*)
(* EXIT the routine IF it was executed the 10 seconds which is equal to 0.04 degrees accuracy *)
IF T_PLC_MS() - last < 10000 THEN RETURN; END_IF;
last := T_PLC_MS();

(* calculate the angles *)
N := DWORD_TO_REAL(DT_TO_DWORD(utc) - 946728000)/86400;
LA := RAD(latitude);
SLA := SIN(LA);
CLA := COS(LA);
LO := Rad(longitude);
L := modR(280.460 + 0.9856474 * N,360);
G := Rad(modR(357.528 + 0.9856003 * N,360));
K := Rad(L + 1.915 * SIN(G) + 0.02 * SIN(2*G));
X := Rad(23.439 - 0.0000004 * N);
A := ATAN(COS(X)*TAN(K));
IF COS(K) < 0 THEN A := A + PI1; END_IF;
D := ASIN(SIN(X) * SIN(K));
TA := RAD(MODR(6.697376 + 0.065709825 * DINT_TO_REAL(TRUNC(N - 0.5)) + 0.5 + TOD_TO_REAL(DT_TO_TOD(utc)) * 2.78538333E-7, 24) * 15 + longitude - DEG(A));
CTA := COS(TA);
T1 := CTA*SLA - TAN(D)*CLA;
B := deg(ATAN(SIN(TA)/T1));
IF T1 < 0 THEN B := B + 180; END_IF;
IF B > 180 THEN
	B := B - 180;
ELSIF B < 180 THEN
	B := B + 180;
END_IF;
H := deg(ASIN(COS(D)*CTA*CLA+SIN(D)*SLA));
HR := H + 0.017 / TAN(Rad(H+10.3/(H+5.11)));


(* revision history
hm	1. feb 2007	rev 1.0
	original version

hm	6. jan 2008	rev 1.1
	performance improvements

hm	18. jan 2008	rev 1.2
	further performance improvements
	only calculate once every 10 seconds

hm	16. mar. 2008	rev 1.3
	added type conversion to avoid warnings under codesys 3.0

hm	30. jun. 2008	rev 1.4
	added type conversions to avoid warnings under codesys 3.0

*)
END_FUNCTION_BLOCK

(* POU SUN_TIME, ST *)
FUNCTION_BLOCK SUN_TIME
VAR_INPUT
	latitude : REAL;				(* latitude of geographical position  *)
	longitude : REAL;				(* longitude of geographical position  *)
	utc : DT;						(*	world time				*)
END_VAR
VAR_OUTPUT
	sun_midday : TOD;			(*	astrological midday in hours when sun stand at south direction	*)
	sun_rise : TOD;				(*	sun rise for current day in local time *)
	sun_set : TOD;				(*	sun set for current day in local time *)
	sun_declination : REAL;		(*	sun declination at midday in degrees	*)
END_VAR
VAR
	T: INT;							(* day in the year   *)
	DK: REAL;						(* sun declination at midday *)
	delta: REAL;					(* delta from midday for sunrise and sunset  *)
	h: REAL;
	B: REAL;
	offset : REAL;
	l15: REAL;
	dat: DATE;
	last_dat: DATE;
END_VAR

(*
version 1.4	17. jan 2008
programmer 	hugo
tested by	tobias

this FUNCTION block calculates the sun rise, sun set, sun offset at midday sun declination for a given date 
for performance reasons the algorithm has been simplified and is accurate within a few minutes only 
the times are calculated in utc and have to be corrected for the given time zone
this correction is not done within sun_time because it would be a problem on days where dst is enabled or disabled


*)
dat := DT_TO_DATE(utc);
IF dat = last_dat THEN RETURN; END_IF;
last_dat := dat;
l15 := longitude * 0.0666666666666;
B := latitude * 0.0174532925199433;
h := -0.0145;
T := day_of_year(dat);
offset := -0.1752 * SIN(0.033430*T + 0.5474) - 0.1340*SIN(0.018234*T - 0.1939);
sun_midday := hour_to_tod(12 + Offset - l15);
DK := 0.40954 * SIN(0.0172 * (T-79.35));
sun_declination := deg(DK);
delta := 12*ACOS((SIN(h) - SIN(B) * SIN(DK)) / (COS(B) * COS(DK))) * 0.318309886;
sun_rise := hour_to_tod(12 - delta - Offset - l15);
sun_set := hour_to_tod(12 + delta - Offset - l15);

(* revision history

rev 1.1	hm	20.1.2007
	deleted unused variables sun_riseR and sun_setR

rev 1.2 hm 17.4.2007
	corrected error while sun:midday would not be corrected for longitude.

rev 1.3	hm	6. jan 2008
	performance improvements

rev	1.4 hm	17. jan 2008
	calculation is now only performed once a day
*)
END_FUNCTION_BLOCK

(* POU SWAP_BYTE, ST *)
FUNCTION SWAP_BYTE : WORD
VAR_INPUT
	IN : WORD;
END_VAR
VAR
END_VAR

(*
version 1.0	4 feb 2008
programmer 	hugo
tested by		tobias

This function swaps the high and low byte of the word in.

*)
Swap_Byte := ROL(in,8);


(* revision history
hm		4. feb 2008	rev 1.0
	original version

*)
END_FUNCTION

(* POU SWAP_BYTE2, ST *)
FUNCTION SWAP_BYTE2 : DWORD
VAR_INPUT
	IN : DWORD;
END_VAR
VAR
END_VAR

(*
version 1.0	4 feb 2008
programmer 	hugo
tested by		tobias

This function reverses the byte order in the dword.

*)
Swap_Byte2 := (ROR(in,8) AND 16#FF00FF00) OR (ROL(in,8) AND 16#00FF00FF);

(* revision history
hm		4. feb 2008	rev 1.0
	original version

*)
END_FUNCTION

(* POU SWITCH_I, ST *)
FUNCTION_BLOCK SWITCH_I
VAR_INPUT
	set : BOOL;
	in : BOOL;
	rst : BOOL;
END_VAR
VAR_INPUT CONSTANT
	T_debounce : TIME := T#10ms;
	T_reconfig : TIME := T#1s;
	T_on_max : TIME := T#0h;
END_VAR
VAR_OUTPUT
	Q : BOOL := 0;
END_VAR
VAR
	state : BYTE := 0;
	edge : BOOL := 0;
	r_edge : BOOL := 0;
	T_on : TIME;
	tx: TIME;
END_VAR

(*
version 1.1	15 sep 2007
programmer 	oscat
tested by		tobias

this is an intelligent switch interface which has an autodetect feature for in and it will detect the type of switch connected automatically
the input can be connected to low active pulses, high active pulses and on/off switch.
it will automatically adjust to the correct type without manual adjustment
a configurable debounce timer will debounce input signals
if t_on_max is set to anything other then 0 the output will be turned off after the max on time is reached.

*)
(* read system time *)
tx := DWORD_TO_TIME(T_PLC_MS());

(* asynchronous set and reset first *)
IF set AND NOT rst THEN
	Q := 1;
	T_on := tx;
ELSIF rst THEN
	Q := 0;
(* check FOR input edge AND start debounce timer *)
ELSIF (in XOR edge) AND NOT (state = 1) THEN
	state := 1;
	T_on := Tx;
(* edge was detected and debounce time elapsed *)
ELSIF (state = 1) AND (Tx - t_debounce >= T_on) THEN
	state := 2;
	(* react on rising or falling edge depending on r_edge *)
	IF r_edge XOR in THEN Q := NOT Q; END_IF;
(* wait for T_reconfig and adjust r_edge *)
ELSIF state = 2 AND Tx - t_reconfig >= T_on THEN
	r_edge := in;
END_IF;
IF Q AND T_on_max > t#0ms AND Tx >= T_on + T_on_max THEN
	Q := FALSE;
END_IF;
edge := in;

(* revision history

hm	4 aug 2006	rev 1.0
	original version

hm	15.9.2007	rev 1.1
	replaced Time() with T_PLC_MS for compatibility and performance reasons

*)
END_FUNCTION_BLOCK

(* POU SWITCH_X, ST *)
FUNCTION_BLOCK SWITCH_X
VAR_INPUT
	IN1 : BOOL;
	IN2 : BOOL;
	IN3 : BOOL;
	IN4 : BOOL;
	IN5 : BOOL;
	IN6 : BOOL;
END_VAR
VAR_OUTPUT
	Q1 : BOOL;
	Q2 : BOOL;
	Q3 : BOOL;
	Q4 : BOOL;
	Q5 : BOOL;
	Q6 : BOOL;
	Q31 : BOOL;
	Q41 : BOOL;
	Q51 : BOOL;
	Q61 : BOOL;
	Q32 : BOOL;
	Q42 : BOOL;
	Q52 : BOOL;
	Q62 : BOOL;
END_VAR
VAR_INPUT CONSTANT
	t_debounce : TIME := t#50ms;
END_VAR
VAR
	init : BOOL;
	T1, T2, T3, T4, T5, T6 : TOF;
	tx: TIME;
	x1: BOOL;
	x2: BOOL;
	E1, E2 : BOOL;
END_VAR

(*
version 1.0	15 Feb 2007
programmer 	oscat
tested by		tobias

*)
(* initialize on startup *)
IF NOT init THEN
	init := TRUE;
	IF t_debounce < t#50ms THEN tx := t#50ms; ELSE tx := t_debounce; END_IF;
	T1(PT := Tx);
	T2(PT := Tx);
	T3(PT := Tx);
	T4(PT := Tx);
	T5(PT := Tx);
	T6(PT := Tx);
ELSE
	Q1 := FALSE;
	Q2 := FALSE;
	Q3 := FALSE;
	Q4 := FALSE;
	Q5 := FALSE;
	Q6 := FALSE;
	Q31 := FALSE;
	Q41 := FALSE;
	Q51 := FALSE;
	Q61 := FALSE;
	Q32 := FALSE;
	Q42 := FALSE;
	Q52 := FALSE;
	Q62 := FALSE;
END_IF;

(* read inputs and debounce *)
	T1(IN := IN1);
	T2(IN := IN2);
	T3(IN := IN3);
	T4(IN := IN4);
	T5(IN := IN5);
	T6(IN := IN6);

(* detect edge of IN1 and IN2 *)
IF t1.Q AND NOT E1 THEN X1 := TRUE; END_IF;
IF t2.Q AND NOT E2 THEN X2 := TRUE; END_IF;

IF t1.Q THEN
	IF t3.q THEN
		q31 := TRUE;
		X1 := FALSE;
	ELSIF t4.q THEN
		q41 := TRUE;
		X1 := FALSE;
	ELSIF t5.q THEN
		q51 := TRUE;
		X1 := FALSE;
	ELSIF t6.q THEN
		q61 := TRUE;
		X1 := FALSE;
	END_IF;
ELSIF t2.Q THEN
	IF t3.q THEN
		q32 := TRUE;
		X2 := FALSE;
	ELSIF t4.q THEN
		q42 := TRUE;
		X2 := FALSE;
	ELSIF t5.q THEN
		q52 := TRUE;
		X2 := FALSE;
	ELSIF t6.q THEN
		q62 := TRUE;
		X2 := FALSE;
	END_IF;
(* in1 was active alone *)
ELSIF NOT T1.Q AND E1 AND X1 THEN
	Q1 := TRUE;
	X1 := FALSE;
ELSIF NOT T2.Q AND E2 AND X2 THEN
	Q2 := TRUE;
	X2 := FALSE;
ELSIF T3.Q THEN
	Q3 := TRUE;
ELSIF T4.Q THEN
	Q4 := TRUE;
ELSIF T5.Q THEN
	Q5 := TRUE;
ELSIF T6.Q THEN
	Q6 := TRUE;
END_IF;

(* save state of in1 and in2 *)
E1 := T1.Q;
E2 := T2.Q;
END_FUNCTION_BLOCK

(* POU TANH, ST *)
FUNCTION TANH : REAL
VAR_INPUT
	X : REAL;
END_VAR
VAR
END_VAR


(*
version 1.2	10. mar 2008
programmer 	hugo
tested by	tobias

this function calculates the tangens hyperbolicus

*)
IF X > 20 THEN
	tanH := 1;
ELSIF X < -20 THEN
	tanH := -1;
ELSE
	tanH := 1 - 2 / (EXP(2 * x) + 1);
END_IF;

(* revision hisdtory
hm		12.1.2007		rev 1.0
	original version

hm		1.12.2007		rev 1.1
	changed code to improve performance

hm		10. mar 2008	rev 1.2
	corrected an error in formula
	extended range of valid inputs to +/- INV
*)
END_FUNCTION

(* POU TANK_LEVEL, ST *)
FUNCTION_BLOCK TANK_LEVEL
VAR_INPUT
	LEVEL : BOOL;
	LEAK : BOOL;
	ACLR : BOOL;
END_VAR
VAR_INPUT CONSTANT
	MAX_VALVE_TIME : TIME := T#0s;
	LEVEL_DELAY_TIME : TIME := T#0s;
END_VAR
VAR_OUTPUT
	VALVE : BOOL;
	ALARM : BOOL;
	STATUS : BYTE;
END_VAR
VAR
	cx : ACTUATOR_COIL;
	tn : TON;
	tl : TONOF;
	open: BOOL;
END_VAR


(*
version 1.0	27 feb 2007
programmer 	hugo
tested by		tobias

*)
(* preprocess the level information *)
tl(in := level, T1 := level_delay_time, T2 := level_delay_time);
open := tl.Q;

(* start logic *)
IF ALARM THEN
	(* check for ACLR if ALARM is present *)
	IF ACLR THEN
		ALARM := FALSE;
		STATUS := 101; (* aclr pressed *)
		cx(in := FALSE);
	END_IF;
	RETURN;
ELSIF LEAK THEN
	(* leakeage detected *)
	cx(in := FALSE);
	ALARM := TRUE;
	STATUS := 1;	(* leakeage error *)
ELSIF open THEN
	(* valve needs to be opened because level is too low *)
	cx(in := TRUE);
	STATUS := 102; (* valve open by low level *)
ELSE
	(* valve needs to be closed *)
	cx(in := FALSE);
	STATUS := 100; (* valve idle *)
END_IF;

(* check if valve is open too long and generate alarm if necessary *)
tn(in := cx.out AND (MAX_VALVE_TIME > T#0s), PT := MAX_VALVE_TIME);
IF tn.Q THEN
	ALARM := TRUE;
	STATUS := 2; (* overtime error *)
	cx(in := FALSE);
END_IF;

(* set output signal *)
VALVE := cx.out;
END_FUNCTION_BLOCK

(* POU TONOF, ST *)
FUNCTION_BLOCK TONOF
VAR_INPUT
	IN : BOOL;
	T1, T2 : TIME;
END_VAR
VAR_OUTPUT
	Q : BOOL;
END_VAR
VAR
	X : TON;
	Y : TOF;
END_VAR

(*
version 1.1	17 sep 2007
programmer 	hugo
tested by		tobias

TONOF generated a TON and TOF Delay for the Input N TON (T1) and TOF (T2) can be configured separately
*)
X(IN := IN, PT := T1);
Y(in := X.Q, PT := T2);
Q := Y.Q;

(* revision history
hm	10. dec 2007	rev 1.0
	original version

*)
	
END_FUNCTION_BLOCK

(* POU TC_MS, ST *)
FUNCTION_BLOCK TC_MS
VAR_INPUT
END_VAR
VAR_OUTPUT
	TC : DWORD;
END_VAR
VAR
	init: BOOL;
	tx: DWORD;
	last: DWORD;
END_VAR

(*
	version 1.0	13 mar 2008
	programmer 	hugo
	tested by		tobias

TC_MS delivers the time it was last called on the output TC in Milliseconds.

*)
(* read system timer *)
tx := T_PLC_MS();

IF NOT init THEN
	init := TRUE;
	TC := 0;
ELSE
	tc := tx - last;
END_IF;
last := tx;

(* revision history
hm		13. mar. 2008	rev 1.0
	original version

*)
END_FUNCTION_BLOCK

(* POU TC_US, ST *)
FUNCTION_BLOCK TC_US
VAR_INPUT
END_VAR
VAR_OUTPUT
	TC : DWORD;
END_VAR
VAR
	init: BOOL;
	tx: DWORD;
	last: DWORD;
END_VAR

(*
	version 1.0	13 mar 2008
	programmer 	hugo
	tested by		tobias

TC_US delivers the time it was last called on the output TC in Microseconds.

*)
(* read system timer *)
tx := T_PLC_US();

IF NOT init THEN
	init := TRUE;
	TC := 0;
ELSE
	tc := tx - last;
END_IF;
last := tx;

(* revision history
hm		13. mar. 2008	rev 1.0
	original version

*)
END_FUNCTION_BLOCK

(* POU TEMP_EXT, ST *)
FUNCTION_BLOCK TEMP_EXT
VAR_INPUT
	t_ext1 : REAL;
	t_ext2 : REAL;
	t_ext3 : REAL;
	t_ext_config : BYTE := 0;
	dt_in : DT;
END_VAR
VAR_INPUT CONSTANT
	t_ext_min : REAL := -40;
	t_ext_max : REAL := 60;
	t_ext_default : REAL := -10;
	heat_period_start : DATE := D#1970-9-1;
	heat_period_stop : DATE := D#1970-4-30;
	cool_period_start : DATE := D#1970-4-1;
	cool_period_stop : DATE := D#1970-9-30;
	heat_start_temp_day : REAL := 15;
	heat_start_temp_night : REAL := 10;
	heat_stop_temp : REAL := 18;
	cool_start_temp_day : REAL := 26;
	cool_start_temp_night : REAL := 26;
	cool_stop_temp : REAL := 24;
	start_day : TOD := tod#09:00;
	start_night : TOD := tod#21:00;
	cycle_time : TIME := t#10m;
END_VAR
VAR_OUTPUT
	t_ext : REAL;
	heat : BOOL;
	cool : BOOL;
END_VAR
VAR
	tx: TIME;
	last_run: TIME;
	init: BOOL;
	cool_start: DATE;
	cool_stop: DATE;
	heat_start: DATE;
	heat_stop: DATE;
	xdate: DATE;
	day: BOOL;
END_VAR


(*
version 1.1	15 sep 2007
programmer 	hugo
tested by		tobias

temp_ext measures and processes ext temperature and decides if heating or cooling is needed.

 the measurement of t_ext has 3 inputs which can be configured in different ways:
	t_ext_config = 0 means the ext temp is the avg of the 3 external temperatures, this mode is the default mode.
	t_ext_config = 1 means t_ext1 is used.
	t_ext_config = 2 means t_ext1 is used.
	t_ext_config = 3 means t_ext1 is used.
	t_ext_config = 4 means t_ext_default is used.
	t_ext_config = 5 means the lowest of the 3 external temperatures is used.
	t_ext_config = 6 means the higest externnal temperature is used.
	t_ext_config = 7 means the midlle external temperature is used, if there are only two working, the lowest is used.
	in any config mode, an external temperature higher then t_ext_max or lower then t_ext_min is ignored to prevent from temperatures caused by broken sensors or wires.
	if no external temperature is available, a default value (t_ext_default) is used.
	if you have only one external sensor, connect the 3 inputs to the same sensor, or select the right input with t_ext_config.

heating or cooling is enabled during heating / cooling period when the day or night start temperature is reached for at least the specified delay time and will be disabled after the stop temperature is reached. 
t_ext output can be used by other modules to determine the correct system temperature for heating or cooling.

*)
IF NOT init THEN
	init := TRUE;
	heat_start := set_Date(1972,month(heat_period_start),day_of_month(heat_period_start));
	heat_stop := set_Date(1972,month(heat_period_stop),day_of_month(heat_period_stop));
	cool_start := set_Date(1972,month(cool_period_start),day_of_month(cool_period_start));
	cool_stop := set_Date(1972,month(cool_period_stop),day_of_month(cool_period_stop));
END_IF;

(* read system time *)
tx := DWORD_TO_TIME(T_PLC_MS());

(* for efficiency exit isf this program has been executed less then 1min ago *)
IF tx - last_run < cycle_time THEN RETURN; END_IF;

(* calculate frequently used variables *)
xdate := set_Date(1972,month(DT_TO_DATE(dt_in)),day_of_month(DT_TO_DATE(dt_in)));
day := DT_TO_TOD(dt_in) >= start_day AND  DT_TO_TOD(dt_in) < start_night;

(* read the correct external temperature depending on the t_ext_config setting *)
t_ext := multi_in(t_ext1, t_ext2, t_ext3, t_ext_default, t_ext_min, t_ext_max, t_ext_config);

(* dtermine heating *)
IF (heat_start <= heat_stop AND xdate >= heat_start AND xdate <= heat_stop) OR (heat_start > heat_stop AND (xdate >= heat_start OR xdate <= heat_stop)) THEN
	(* heating period id true check for temperature *)
	IF day AND t_ext <= heat_start_temp_day THEN
		heat := TRUE;
	ELSIF NOT day AND t_ext <= heat_start_temp_night THEN
		heat := TRUE;
	ELSIF t_ext >= heat_stop_temp THEN
		heat := FALSE;
	END_IF;
ELSE
	heat := FALSE;
END_IF;

(* dtermine cooling *)
IF (cool_start <= cool_stop AND xdate >= cool_start AND xdate <= cool_stop) OR (cool_start > cool_stop AND (xdate >= cool_start OR xdate <= cool_stop)) THEN
	(* cooling period is true check for temperature *)
	IF day AND t_ext >= cool_start_temp_day THEN
		cool := TRUE;
	ELSIF NOT day AND t_ext >= cool_start_temp_night THEN
		cool := TRUE;
	ELSIF t_ext <= cool_stop_temp THEN
		cool := FALSE;
	END_IF;
ELSE
	cool := FALSE;
END_IF;

last_run := tx;

(* revision history
hm	6 dec 2006		rev 1.0
	original version

hm	15.9.2007		rev 1.1
	replaced Time() with T_PLC_MS for compatibility and performance reasons

*)
END_FUNCTION_BLOCK

(* POU TEMP_NI, ST *)
FUNCTION TEMP_NI : REAL
VAR_INPUT
	Res : REAL;
	R0 : REAL;
END_VAR
VAR
END_VAR

(*
version 1.4	6. Jan 2008
programmer 	hugo
tested by		tobias

this function returns the temperature for a nickel sensor in a range from -60..+180 °C *)
Temp_NI := (SQRT(0.30085225 - 2.66E-3 * (R0 - Res)) - 0.5485) * 751.8796992;

(*Temp_NI := 60;
WHILE step > accuracy DO
	IF Res_NI(Temp_NI,R0) < res THEN Temp_NI := Temp_NI + step; ELSE Temp_NI := Temp_NI - step; END_IF;
	step := step / 2;
END_WHILE;
*)
(* code before rev 1.3
Temp_NI := -60.0;
WHILE step > accuracy DO
	(* test if result greater or less *)
	IF Res_NI(Temp_NI + step,R0) < res THEN Temp_NI := Temp_NI + step; END_IF;
	step := step / 2;
END_WHILE;
*)

(* revision history

rev 1.1 	hm 24.1.2007	
	deleted unused variable A, B, C

rev 1.2		hm 10.9.2007
	changed accuracy to 0.02 degrees to improove performace

hm 17. 12 2007		rev 1.3
	improovements for better performance and higher accuracy

hm	6. jan 2008		rev 1.4
	further performance improvement
*)
END_FUNCTION

(* POU TEMP_PT, ST *)
FUNCTION TEMP_PT : REAL
VAR_INPUT
	Res : REAL;
	R0 : REAL;
END_VAR
VAR CONSTANT
	A : REAL := 3.9083E-3 ;
	B : REAL := -5.775E-7;
	accuracy : REAL := 0.02;
END_VAR
VAR
	step: REAL := 50.0;
	X: REAL;
	Y: REAL;
	t1: REAL;
END_VAR

(*
version 1.5	5. jan 2008
programmer 	hugo
tested by		tobias

this function returs the temperature for a platinum sensor for a range from -200..+850 °C *)
X := A * R0;
Y := B * R0;
IF Res >= R0 THEN
	t1 := X*X-4*Y*(R0-Res);
	IF t1 < 0 THEN
		Temp_PT := 10000;
	ELSE
		Temp_PT := (-X + SQRT(t1)) / (2 * Y);
	END_IF;
ELSE
	(* since the formula cannot be solved this is a successive approximation *)
	Temp_PT := -100.0;
	WHILE step > accuracy DO
		(* test if result greater or less *)
		IF Res_PT(Temp_PT,R0) < res THEN Temp_PT := Temp_PT + step; ELSE Temp_PT := Temp_PT - step; END_IF;
		step := step * 0.5;
	END_WHILE;
END_IF;

(* revision history

rev 1.1 hm 24.1.2007	
	deleted unused variable C

rev 1.2 hm 10.9.2007
	reduced accuracy to 0.02 to shorten execution time

rev 1.3	hm	2. dec 2007
	changed code for better performance

rev	1.4	hm	23. dec 2007
	avoid a negative square root if input values are wrong

rev 1.5 hm	5. jan 2008
	replaced / 2 with * 0.5 for better performance
*)
END_FUNCTION

(* POU TEMP_SI, ST *)
FUNCTION TEMP_SI : REAL
VAR_INPUT
	Res : REAL;
	RS : REAL;
	TS : REAL;
END_VAR
VAR CONSTANT
END_VAR
VAR
END_VAR

(*
version 1.4	6. jan 2008
programmer 	hugo
tested by		tobias

this function returs the temperature for a silicon sensor for a range from -60..+180 °C
for example KTY10 RS at TS normally 25 °C
*)
Temp_SI := (-7.64E-3 + SQRT(Res/RS* 6.64E-5 - 0.803E-5)) * 30120.48193 + TS;

(* code before rev 1.3
Temp_SI := -60;
WHILE step > accuracy DO
	(* test if result greater or less *)
	IF Res_SI(Temp_SI + step,RS,TS) < Res THEN Temp_SI := Temp_SI + step; END_IF;
	step := step / 2;
END_WHILE;
*)

(* revision history

hm 24.1.2007		rev 1.1
	the function would only work for TS = 25, now it works for other values of ts.

hm 10.9.2007		rev 1.2
	changed the function to use successive approcimation to avoid an error generated by a sqrt from a negative result.
	changed accuracy to 0.02 degrees to shorten execution time

hm 17. 12 2007		rev 1.3
	improovements for better performance

hm	6. jan 2008		rev 1.4
	further performance improvement
*)
END_FUNCTION

(* POU TEMPERATURE, ST *)
FUNCTION_BLOCK TEMPERATURE
VAR_INPUT
	K : REAL;
	C : REAL := -273.15;
	F : REAL := -459.67;
	Re : REAL := -218.52;
	Ra : REAL := 0;
END_VAR
VAR_OUTPUT
	YK : REAL;
	YC : REAL;
	YF : REAL;
	YRe : REAL;
	YRa : REAL;
END_VAR
VAR
END_VAR

(*
version 1.0	21 feb 2008
programmer 	hugo
tested by	oscat

this function converts different temperature units
any unused input can simply be left open.
different inputs connected at the same time will be added up.

*)
YK := K + (C + 273.15) + (F + 459.67) * 0.555555555555 + (Re * 1.25 + 273.15) + (Ra * 0.555555555555);
YC := YK -273.15;
YF := YK * 1.8 - 459.67;
YRe := (YK - 273.15) * 0.8;
YRa := YK * 1.8;


(* revision history
hm	21. feb. 2008	rev 1.0
	original version

*)
END_FUNCTION_BLOCK

(* POU TICKER, ST *)
FUNCTION_BLOCK TICKER

VAR_INPUT
	N : INT;
	PT : TIME;
END_VAR

VAR_IN_OUT
	Text : STRING(STRING_LENGTH);
END_VAR

VAR_OUTPUT
	Display : STRING(STRING_LENGTH);
END_VAR
VAR
	delay : TP;
	step : INT;
END_VAR

(*
version 1.2	29. mar. 2008
programmer 	hugo
tested by		tobias

Ticker sends a substring of text with length N every TD Milliseconds to generate a ticker. 

*)
(* generate next ticker when delay is low *)
IF N < LEN(text) THEN
	IF NOT delay.Q THEN
		(* increase step for next tick *)
		step := step + 1;
		IF step > LEN(text) THEN step := 1; END_IF;
		(* extract dispay from text *)
		display := MID(text, N, step);
		(* set delay timer for next tick *)
		delay(in := TRUE, PT := PT);
	ELSE;
		(* execute delay timer *)
		delay(in := FALSE);
	END_IF;
ELSE
	display := text;
END_IF;
(* revision history
hm	4. dec. 2007	rev 1.0
	original version

hm	15. dec. 2007	rev 1.1
	step now starts at 1 instaed of 0

hm	29. mar. 2008	rev 1.2
	changed STRING to STRING(STRING_LENGTH)
*)
END_FUNCTION_BLOCK

(* POU TIMER_2, ST *)
FUNCTION_BLOCK TIMER_2
VAR_INPUT
	DT_in : DT;
	start : TOD;
	duration : TIME;
	mode : BYTE;
	holiday : BOOL;
END_VAR
VAR_OUTPUT
	Q : BOOL;
END_VAR
VAR
	last_check : TIME := T#0s;
	dat : DATE;
	daytime : TOD;
	activation: TIME;
	tx: TIME;
	enabled: BOOL;
	wday: INT;
	init: BOOL;
END_VAR

VAR RETAIN
	run_date : DATE;
END_VAR

(*
version 1.2	15 sep 2007
programmer 	oscat
tested by		tobias

this timer generated programmabe output pulses per day, week, month and so on.
the mode input determines on which days the timer will be active.
	mode = 0			never
	mode = 1..7		monday .. sunday
	mode = 11			every day
	mode = 12			every second day
	mode = 13			every 3rd day
	mode = 14			every 4th day
	mode = 15			every 5th day
	mode = 16 		every 6th day
	mode = 20			only monday - friday
	mode = 21			only sat - sunday
	mode = 22			workdays only
	mode = 23			holidays and weekend
	mode = 24			holidays only
	mode = 25			every 1st day of the month
	mode = 26			every last day of the month
	mode = 27			every 31 of december
	mode = 28			every 1st of january

a holiday input can be used to supply holiday information to the module.
*)
(* read system time *)
tx := DWORD_TO_TIME(T_PLC_MS());

IF NOT init THEN
	init := TRUE;
	last_check := tx - t#100ms;
END_IF;

(* for performance resons exit if execution is not necessary *)
IF tx - last_check <= T#100ms THEN RETURN; END_IF;

(* calculate temp variables *)
dat := DT_TO_DATE(dt_in);
daytime := DT_TO_TOD(dt_in);
wday := weekday(dat);

(* calculate if any action is necessary today *)
enabled := FALSE;
CASE mode OF
1..7:	(* mondays to fridays *)
	IF wday = mode THEN enabled := 1; END_IF;
11:	(* every day *)
	enabled := TRUE;
12..16:	(* every nth day *)
	IF (TRUNC(DATE_TO_DWORD(dat)/86400)) MOD (mode - 10) = 0 THEN enabled := 1; END_IF;
20:	(* monday - friday *)
	IF wday <= 5 THEN enabled := TRUE; END_IF;
21:	(* saturday and sunday *)
	IF wday > 5 THEN enabled := TRUE; END_IF;
22: (* workdays only *)
	IF wday <= 5 AND NOT holiday THEN enabled := TRUE; END_IF;
23:	(* holidays and weekends *)
	IF wday > 5 OR holiday THEN enabled := TRUE; END_IF;
24:	(* holidays only *)
	enabled := holiday;
25:	(* 1st day of the month *)
	IF day_of_month(dat) = 1 THEN enabled := TRUE; END_IF;
26:	(* last day of month *)
	IF day_of_month(dat + t#1d) = 1 THEN enabled := TRUE; END_IF;
27:	(* 31st of december *)
	IF day_of_month(dat) = 31 AND month(dat) = 12 THEN enabled := TRUE; END_IF;
28:	(* 1st of january *)
	IF day_of_year(dat) = 1 THEN enabled := TRUE; END_IF;
END_CASE;

(* set or reset output if necessary *)
IF enabled AND NOT Q AND daytime >= start AND run_date <> dat THEN
	Q := 1;
	activation := tx;
	run_date := dat;
ELSIF Q AND tx - activation >= duration THEN
	Q := 0;
END_IF;
last_check := Tx;


(* revision history
hm 22.2.2007		rev 1.1
	changed VAR RETAIN PERSISTENT to VAR RETAIN for better compatibility
	wago lon contollers do not support persisitent

hm	15.9.2007		rev 1.2
	replaced Time() with T_PLC_MS for compatibility and performance reasons
 
*)
END_FUNCTION_BLOCK

(* POU TIMER_EVENT_DECODE, ST *)
FUNCTION TIMER_EVENT_DECODE : TIMER_EVENT
VAR_INPUT
	EVENT : STRING(STRING_LENGTH);
END_VAR
VAR
	pos: INT;
	start : INT;
	stop: INT;
	pt : POINTER TO ARRAY[1..255] OF BYTE;
	step: INT;
	tmp : STRING(60);
END_VAR



(*
version 1.0	17. jun 2008
programmer 	hugo
tested by	oscat

STRING_TO_TIMER_EVENT converts a string to a timer event structure.

*)
(* a timer event is specified as follows:
	$typ;ch;day;start;duration;land;lor#
$ 		= start of definition
typ 	= type of definition	(number)
channel	= channel number		(number)
day 	= day number			(number)
start	= start time			(time of day)
duration= duration of event		(time)
land	= mask for output AND	(8bit value)
lor		= mask for ourput OR	(8bit value)
#		= end of definition
*)

(* check for start and ending character *)
IF (LEFT(event,1) <> '<') AND (RIGHT(event,1) <> '>') THEN RETURN; END_IF;
stop := LEN(event);
pt := ADR(event);
start := 2;

(* parse the string for next ; *)
FOR pos := 2 TO stop DO
	IF pt^[pos] = 59 OR pt^[pos] = 62 THEN
		tmp := MID(event, pos - start, start);
		CASE step OF
			0:	(* read type *)
				TIMER_EVENT_DECODE.typ := FSTRING_TO_BYTE(tmp);

			1:	(* read channel *)
				TIMER_EVENT_DECODE.channel := FSTRING_TO_BYTE(tmp);

			2:	(* read day *)
				IF IS_CC(tmp,'0123456789abcdefABCDEF#') THEN
					TIMER_EVENT_DECODE.day := FSTRING_TO_BYTE(tmp);
				ELSIF TIMER_EVENT_DECODE.typ = 2 THEN
					TIMER_EVENT_DECODE.DAY := FSTRING_TO_WEEK(tmp);
				ELSE
					TIMER_EVENT_DECODE.DAY := INT_TO_BYTE(FSTRING_TO_WEEKDAY(tmp));
				END_IF;

			3:	(* read start *)
				TIMER_EVENT_DECODE.start := STRING_TO_TOD(tmp);

			4:	(* read duaration *)
				TIMER_EVENT_DECODE.duration := STRING_TO_TIME(tmp);

			5:	(* read land *)
				TIMER_EVENT_DECODE.land := FSTRING_TO_BYTE(tmp);

			6:	(* read lor *)
				TIMER_EVENT_DECODE.LOR := FSTRING_TO_BYTE(tmp);
		END_CASE;
		start := pos + 1;
		step := step + 1;
	END_IF;
END_FOR;




(* revision history
hm	17. jun 2008		rev 1.0
	original version

*)
END_FUNCTION

(* POU TIMER_P4, ST *)
FUNCTION_BLOCK TIMER_P4
VAR_INPUT
	DTIME : DT;
	TREF_0 : TOD;
	TREF_1 : TOD;
	HOLY : BOOL;
	L0, L1, L2, L3 : BOOL;
	OFS : INT;
	DIS : BOOL;
	MAN : BOOL;
	MI : BYTE;
	RST : BOOL;
END_VAR
VAR_IN_OUT
	PROG : ARRAY[0..array_max] OF TIMER_EVENT;
END_VAR
VAR_OUTPUT
	Q0, Q1, Q2, Q3 : BOOL;
	STATUS : BYTE;
END_VAR
VAR CONSTANT
	array_max : INT := 63;
	channel_max : INT := 3;
END_VAR
VAR
	pos : INT;
	last_execute: DT;
	current_day : DWORD;
	timer: ARRAY[0..channel_max] OF TOF;
	mask: BYTE;
	ma : ARRAY[0..channel_max] OF BYTE;
	mo : ARRAY[0..channel_max] OF BYTE;
	channel: INT;
	tx: TOD;
END_VAR


(*
version 1.0	17. jun 2008
programmer 	hugo
tested by	oscat

TIMER_P4 is a programmable universal timer.


*)
(* for performance reasons we only execute the code at the beginning of a new second
	we cannot compare the dtime directly because a daylight savings time switch might have happened
	therefore we need to compare the seconds and minutes of the dtime only 
	if we would compare seconds only the module would be in troulbe when its only called every minute 
	with this code the module is called every start of a new second *)

IF RST THEN
	last_execute := DT#1970-1-1-00:00;
	FOR pos := 0 TO ARRAY_MAX DO
		IF (PROG[pos].CHANNEL >= OFS) AND (PROG[pos].CHANNEL - OFS < 0) THEN PROG[pos].LAST := 0; END_IF;
	END_FOR;
	FOR pos := 0 TO channel_max DO
		timer[pos](pt := t#0s);
	END_FOR;
	status := 100;
ELSIF dtime <> last_execute THEN
	(* prepare the logical input mask to be used later *)
	mask := 255;
	mask.0 := L0;
	mask.1 := L1;
	mask.2 := L2;
	mask.3 := L3;
	(* save the actual second for next execution test *)
	last_execute := DTIME;
	current_day := DINT_TO_DWORD(DAY_OF_DATE(DT_TO_DATE(Dtime)));
	pos := 0;
	WHILE pos <= ARRAY_MAX DO
		channel := prog[pos].CHANNEL - OFS;
		IF (prog[pos].TYP > 0) AND (channel >= 0) AND (channel <= channel_max) THEN
			ma[channel] := prog[pos].LAND;
			mo[channel] := prog[pos].LOR;
			CASE prog[pos].TYP OF
				1:	(* daily event *)
					IF (DT_TO_TOD(dtime) >= prog[pos].START) AND (current_day <> prog[pos].last) THEN
						prog[pos].LAST := current_day;	(* make sure we only execute once a day *)
						timer[MIN(channel_max, prog[pos].CHANNEL - OFS)](in := NOT DIS, PT := prog[pos].DURATION);
					END_IF;
					status := 101;
				2: 	(* event by selected weekdays *)
					IF (DT_TO_TOD(dtime) >= prog[pos].START) AND (current_day <> prog[pos].last) AND ((SHR(BYTE#128, WEEKDAY(DT_TO_DATE(Dtime))) AND prog[pos].DAY) > 0) THEN
						prog[pos].LAST := current_day;	(* make sure we only execute once a day *)
						timer[MIN(channel_max, prog[pos].CHANNEL - OFS)](in := NOT DIS, PT := prog[pos].DURATION);
					END_IF;
					status := 102;
				3:	(* event every N days *)
					IF (DT_TO_TOD(dtime) >= prog[pos].START) AND (current_day <> prog[pos].last) AND (prog[pos].LAST + prog[pos].DAY >= current_day) THEN
						prog[pos].LAST := current_day;	(* make sure we only execute once a day *)
						timer[MIN(channel_max, prog[pos].CHANNEL - OFS)](in := NOT DIS, PT := prog[pos].DURATION);
					END_IF;
					status := 103;
				10:	(* weekly event exactly once a week the weekday is specified in day, 1= mo *)
					IF (DT_TO_TOD(dtime) >= prog[pos].START) AND (current_day <> prog[pos].last) AND WEEKDAY(DT_TO_DATE(DTIME)) = prog[pos].DAY THEN
						prog[pos].LAST := current_day;	(* make sure we only execute once a day *)
						timer[MIN(channel_max, prog[pos].CHANNEL - OFS)](in := NOT DIS, PT := prog[pos].DURATION);
					END_IF;
					status := 110;
				20:	(* monthly event *)
					IF (DT_TO_TOD(dtime) >= prog[pos].START) AND (current_day <> prog[pos].last) AND DAY_OF_MONTH(DT_TO_DATE(DTIME)) = prog[pos].DAY THEN
						prog[pos].LAST := current_day;	(* make sure we only execute once a day *)
						timer[MIN(channel_max, prog[pos].CHANNEL - OFS)](in := NOT DIS, PT := prog[pos].DURATION);
					END_IF;
					status := 120;
				21:	(* event on last day of month *)
					IF (DT_TO_TOD(dtime) >= prog[pos].START) AND (current_day <> prog[pos].last) AND (DT_TO_DATE(DTIME) = MONTH_END(DT_TO_DATE(dtime))) THEN
						prog[pos].LAST := current_day;	(* make sure we only execute once a day *)
						timer[MIN(channel_max, prog[pos].CHANNEL - OFS)](in := NOT DIS, PT := prog[pos].DURATION);
					END_IF;
					status := 121;
				30:	(* yearly event on a specific day specified in day *)
					IF (DT_TO_TOD(dtime) >= prog[pos].START) AND (current_day <> prog[pos].last) AND DAY_OF_YEAR(DT_TO_DATE(DTIME)) = prog[pos].DAY THEN
						prog[pos].LAST := current_day;	(* make sure we only execute once a day *)
						timer[MIN(channel_max, prog[pos].CHANNEL - OFS)](in := NOT DIS, PT := prog[pos].DURATION);
					END_IF;
					status := 130;
				31:	(* event on last day of year *)
					IF (DT_TO_TOD(dtime) >= prog[pos].START) AND (current_day <> prog[pos].last) AND (DT_TO_DATE(DTIME) = YEAR_END(YEAR(DT_TO_DATE(dtime)))) THEN
						prog[pos].LAST := current_day;	(* make sure we only execute once a day *)
						timer[MIN(channel_max, prog[pos].CHANNEL - OFS)](in := NOT DIS, PT := prog[pos].DURATION);
					END_IF;
					status := 131;
				40:	(* event on leap days *)
					IF (DT_TO_TOD(dtime) >= prog[pos].START) AND (current_day <> prog[pos].last) AND LEAP_DAY(DT_TO_DATE(dtime)) THEN
						prog[pos].LAST := current_day;	(* make sure we only execute once a day *)
						timer[MIN(channel_max, prog[pos].CHANNEL - OFS)](in := NOT DIS, PT := prog[pos].DURATION);
					END_IF;
					status := 140;
				41: (* event on holidays *)
					IF (DT_TO_TOD(dtime) >= prog[pos].START) AND (current_day <> prog[pos].last) AND Holy THEN
						prog[pos].LAST := current_day;	(* make sure we only execute once a day *)
						timer[MIN(channel_max, prog[pos].CHANNEL - OFS)](in := NOT DIS, PT := prog[pos].DURATION);
					END_IF;
					status := 141;
				42: (* event on holidays and weekends *)
					IF (DT_TO_TOD(dtime) >= prog[pos].START) AND (current_day <> prog[pos].last) AND (Holy OR (WEEKDAY(DT_TO_DATE(dtime)) = 6) OR (WEEKDAY(DT_TO_DATE(dtime)) = 7)) THEN
						prog[pos].LAST := current_day;	(* make sure we only execute once a day *)
						timer[MIN(channel_max, prog[pos].CHANNEL - OFS)](in := NOT DIS, PT := prog[pos].DURATION);
					END_IF;
					status := 142;
				43:	(* event on workdays Mo-FR and no holiday *)
					IF (DT_TO_TOD(dtime) >= prog[pos].START) AND (current_day <> prog[pos].last) AND (NOT Holy) AND (WEEKDAY(DT_TO_DATE(dtime)) < 6) THEN
						prog[pos].LAST := current_day;	(* make sure we only execute once a day *)
						timer[MIN(channel_max, prog[pos].CHANNEL - OFS)](in := NOT DIS, PT := prog[pos].DURATION);
					END_IF;
					status := 143;
				50: (* event after reference time *)
					CASE prog[pos].DAY OF
						0:	tx := tref_0;
						1:	tx := tref_1;
					END_CASE;
					IF (DT_TO_TOD(dtime) >= (tx + TOD_TO_TIME(prog[pos].START))) AND (current_day <> prog[pos].last) THEN
						prog[pos].LAST := current_day;	(* make sure we only execute once a day *)
						timer[MIN(channel_max, prog[pos].CHANNEL - OFS)](in := NOT DIS, PT := prog[pos].DURATION);
					END_IF;
					status := 150;
				51:	(* event before reference time *)
					CASE prog[pos].DAY OF
						0:	tx := tref_0;
						1:	tx := tref_1;
					END_CASE;
					IF (DT_TO_TOD(dtime) >= (tx - TOD_TO_TIME(prog[pos].START))) AND (current_day <> prog[pos].last) THEN
						prog[pos].LAST := current_day;	(* make sure we only execute once a day *)
						timer[MIN(channel_max, prog[pos].CHANNEL - OFS)](in := NOT DIS, PT := prog[pos].DURATION);
					END_IF;
					status := 151;
				ELSE
					status := 100;
			END_CASE;
		END_IF;
		pos := pos + 1;
	END_WHILE;
END_IF;

(* since the timers are edge driven we need to reset the timer inputs *)
FOR pos := 0 TO channel_max DO
	timer[pos](IN := FALSE);
END_FOR;

(* set the outputs *)
Q0 := timer[0].Q AND ((ma[0] AND mask) = ma[0]) OR ((mo[0] AND mask) > 0) OR (man AND MI.0);
Q1 := timer[1].Q AND ((ma[1] AND mask) = ma[1]) OR ((mo[1] AND mask) > 1) OR (man AND MI.1);
Q2 := timer[2].Q AND ((ma[2] AND mask) = ma[2]) OR ((mo[2] AND mask) > 2) OR (man AND MI.2);
Q3 := timer[3].Q AND ((ma[3] AND mask) = ma[3]) OR ((mo[3] AND mask) > 3) OR (man AND MI.3);
IF MAN THEN status := 199; END_IF;




(* revision history
hm	17. jun 2008		rev 1.0
	original version

*)
END_FUNCTION_BLOCK

(* POU YEAR_END, ST *)
FUNCTION YEAR_END : DATE
VAR_INPUT
	y : INT;
END_VAR
VAR
END_VAR

(*
version 1.0	15. jun. 2008
programmer 	hugo
tested by	oscat

returs the date of december 31st for the given year  
the function works for dates from 1970 - 2099 

*)
YEAR_END := DWORD_TO_DATE(SHR(INT_TO_DWORD(y+1) * 1461 - 2878173,2)*86400);



(* revision history
hm	15. jun. 2008	rev 1.0
	original version

*)
END_FUNCTION

(* POU TOGGLE, ST *)
FUNCTION_BLOCK TOGGLE
VAR_INPUT
	CLK : BOOL;
	rst : BOOL := FALSE;
END_VAR
VAR_OUTPUT
	Q : BOOL;
END_VAR
VAR
	edge : BOOL;
END_VAR

(*
version 1.0	13 sep 2007
programmer 	hugo
tested by		tobias

toggle flip flop the output changes state with every rising edge of clk.

*)
IF rst THEN
	q := 0;
ELSIF clk AND NOT edge THEN
	Q := NOT Q;
END_IF;
edge := clk;

(* revision history

hm	13.9.2007		rev 1.0
	original version

*)
END_FUNCTION_BLOCK

(* POU TRIANGLE_A, ST *)
FUNCTION TRIANGLE_A : REAL
VAR_INPUT
	S1 : REAL;
	A : REAL;
	S2 : REAL;
	S3 : REAL;
END_VAR
VAR
END_VAR

(*
version 1.1	22. feb 2008
programmer 	hugo
tested by		tobias

triangle_A calculates the Area of a triangle.
if any input is 0 it will be neglected and the are will be calculated from eiter:
two sides and an angle (s1 and S2 and the angle A1) or 3 sides.


*)
IF A = 0 THEN
	triangle_A := SQRT((s1+s2+S3) * (s1+s2-S3) * (S2+S3-S1) * (S3+S1-S2)) * 0.25;
ELSE
	triangle_A := S1 * S2 * SIN(Rad(A)) * 0.5;
END_IF;

(* revision histroy
hm	16. oct 2007	rev 1.0
	original version

hm	22. feb 2008	rev 1.1
	improved performance
*)
END_FUNCTION

(* POU TRIM1, ST *)
FUNCTION TRIM1 : STRING(STRING_LENGTH)
VAR_INPUT
	str : STRING(STRING_LENGTH);
END_VAR
VAR
	pos: INT;
END_VAR

(*
version 1.2	29. mar. 2008
programmer 	hugo
tested by		tobias

the function replaces all multiple blanks within a string by only one blank.
leading and ending blanks will be deleted

*)
TRIM1 := str;
REPEAT
	pos := FIND(trim1,'  ');
	IF pos > 0 THEN TRIM1 := REPLACE(TRIM1,' ',2,pos); END_IF;
UNTIL pos = 0	END_REPEAT;
(* beginning and ending blanks need to be stripped off *)
IF LEFT(trim1,1) = ' ' THEN trim1 := DELETE(trim1,1,1); END_IF;
IF RIGHT(trim1,1) = ' ' THEN trim1 := DELETE(trim1,1,LEN(trim1)); END_IF;


(* revision histroy
hm	4. feb. 2008    rev 1.0
	original release

hm	20. mar. 2008	rev 1.1
	avoid to call replace with pos = 0 because some systems will produce an error

hm	29. mar. 2008	rev 1.2
	changed STRING to STRING(STRING_LENGTH)
*)
END_FUNCTION

(* POU TRIME, ST *)
FUNCTION TRIME : STRING(STRING_LENGTH)
VAR_INPUT
	str : STRING(STRING_LENGTH);
END_VAR
VAR
END_VAR

(*
version 1.0	28. mar. 2008
programmer 	hugo
tested by	tobias

this function deletes all leading and ending blanks of a string.

*)
TRIME := str;
(* beginning blanks need to be stripped off *)
WHILE LEFT(TRIME,1) = ' ' DO
	TRIME := DELETE(TRIME,1,1);
END_WHILE;

(* ending blanks need to be stripped off *)
WHILE RIGHT(TRIME,1) = ' ' DO
	TRIME := DELETE(TRIME,1,LEN(TRIME));
END_WHILE;


(* revision histroy
hm	28. mar. 2008	rev 1.0
	original release

*)
END_FUNCTION

(* POU TUNE, ST *)
FUNCTION_BLOCK TUNE
VAR_INPUT
	SET : BOOL;
	SU, SD : BOOL;
	RST : BOOL;
END_VAR
VAR_INPUT CONSTANT
	SS : REAL := 0.1;
	Limit_L : REAL := 0;
	LIMIT_H : REAL := 100;
	RST_val : REAL := 0;
	SET_val : REAL := 100;
	T1 : TIME := T#500ms;
	T2 : TIME := T#2s;
	S1 : REAL := 2;
	S2 : REAL := 10;
END_VAR
VAR_OUTPUT
	Y : REAL;
END_VAR
VAR
	tx : DWORD;
	start, start2 : DWORD;
	state : INT;
	in : BOOL;
	step : REAL;
	speed : REAL;
	Y_start : REAL;
	Y_start2: REAL;
END_VAR

(*
version 1.1	16. mar 2008
programmer 	hugo
tested by	tobias

tune generates an output signal which is set by input switches.
up to 4 switsches can be used to tune the signal up or down.

*)
(* read system time *)
tx := T_PLC_MS();

IF rst THEN
	Y := RST_val;
	state := 0;
ELSIF set THEN
	Y := SET_val;
	state := 0;
ELSIF state > 0 THEN
	(* key has been pushed state machine operating *)
	(* first read the correct input *)
	IF state = 1 THEN
		(* step up *)
		in := su;
	ELSE
		(* step down *)
		in := sd;
	END_IF;
	(* check for single step operation *)
	IF NOT in AND tx - start <= TIME_TO_DWORD(T1) THEN
		Y := Y_start + step;
		state := 0;
	(* check if fast ramp needs to be generated *)
	ELSIF in AND tx - start >= TIME_TO_DWORD(T2) THEN
		Y := Y_start2 + DWORD_TO_REAL(tx - start2) * s2 / speed;
	(* check if slow ramp needs to be generated *)
	ELSIF in AND tx - start >= TIME_TO_DWORD(T1) THEN
		Y := Y_start + DWORD_TO_REAL(tx - start - TIME_TO_DWORD(T1)) * S1 / speed;
		start2 := tx;
		Y_start2 := Y;
	ELSIF NOT in THEN
		state := 0;
	END_IF;
ELSIF su THEN
	(* slow step up *)
	state := 1;
	start := tx;
	step := ss;
	speed := 1000;
	Y_start := Y;
ELSIF sd THEN
	(* slow step down *)
	state := 2;
	start := tx;
	step := -ss;
	speed := -1000;
	Y_start := Y;
END_IF

(* make sure output does not exceed limits *)
Y := LIMIT(LIMIT_L, Y, LIMIT_H);

(* revision history
hm		3.11.2007		rev 1.0
	original version

hm		16. mar. 2008	rev 1.1
	added type conversions to avoid warnings under codesys 3.0
*)
END_FUNCTION_BLOCK

(* POU TUNE2, ST *)
FUNCTION_BLOCK TUNE2
VAR_INPUT
	SET : BOOL;
	SU, SD : BOOL;
	FU, FD : BOOL;
	RST : BOOL;
END_VAR
VAR_INPUT CONSTANT
	SS : REAL := 0.1;
	FS : REAL := 5;
	Limit_L : REAL := 0;
	LIMIT_H : REAL := 100;
	RST_val : REAL := 0;
	SET_val : REAL := 100;
	TR : TIME := T#500ms;
	S1 : REAL := 2;
	S2 : REAL := 10;
END_VAR
VAR_OUTPUT
	Y : REAL;
END_VAR
VAR
	tx : DWORD;
	start : DWORD;
	state : INT;
	in : BOOL;
	step : REAL;
	speed : REAL;
	Y_start : REAL;
END_VAR

(*
version 1.1	16. mar. 2008
programmer 	hugo
tested by		tobias

tune2 generates an output signal which is set by input switches.
up to 4 switsches can be used to tune the signal up or down.

*)
(* read system time *)
tx := T_PLC_MS();

IF rst THEN
	Y := RST_val;
	state := 0;
ELSIF set THEN
	Y := SET_val;
	state := 0;
ELSIF state > 0 THEN
	(* key has been pushed state machine operating *)
	(* first read the correct input *)
	CASE state OF
		1 :	(* slow up *)
			in := su;
		2 :	(* slow down *)
			in := sd;
		3 :	(* fast up *)
			in := fu;
		4 :	(* fast down *)
			in := fd;
	END_CASE;
	(* check for single step operation *)
	IF NOT in AND tx - start <= TIME_TO_DWORD(TR) THEN
		Y := Y_start + step;
		state := 0;
	(* check if ramp needs to be generated *)
	ELSIF in AND tx - start >= TIME_TO_DWORD(TR) THEN
		Y := Y_start + DWORD_TO_REAL(tx - start - TIME_TO_DWORD(TR)) * speed;
	ELSIF NOT in THEN
		state := 0;
	END_IF;
ELSIF su THEN
	(* slow step up *)
	state := 1;
	start := tx;
	step := ss;
	speed := s1 * 1E-3;
	Y_start := Y;
ELSIF sd THEN
	(* slow step down *)
	state := 2;
	start := tx;
	step := -ss;
	speed := -s1 * 1E-3;
	Y_start := Y;
ELSIF fu THEN
	(* fast step up *)
	state := 3;
	start := tx;
	step := fs;
	speed := s2 * 1E-3;
	y_start := Y;
ELSIF fd THEN
	(* fast step down *)
	state := 4;
	start := tx;
	step := -fs;
	speed := -s2 * 1E-3;
	y_start := Y;
END_IF

(* make sure output does not exceed limits *)
Y := LIMIT(LIMIT_L, Y, LIMIT_H);

(* revision history
hm		3.11.2007		rev 1.0
	original version

hm		16. 3. 2008	rev 1.1
	added type conversions to avoid warnings in codesys 3.0
	improved performance
*)
END_FUNCTION_BLOCK

(* POU URL_DECODE, ST *)
FUNCTION URL_DECODE : STRING(255)
VAR_INPUT
	IN : STRING(255);
END_VAR
VAR
	pos : INT;
	seq : STRING(3);
	new : STRING(1);
END_VAR


(*
version 1.0		27. apr. 2008
programmer 		hugo
tested by		hugo

URL_DECODE checks a string if it contains non reserved characters represented by a % followed with the two digit hex code and converts them to their ascii code.
the non reserved characters are : [A..Z], [a..z], [0..9], -_.~
for example the character sequence '%23' will be converted to '#'.

*)
URL_DECODE := IN;
pos := FIND(URL_DECODE,'%');
WHILE pos > 0 DO
	seq := MID(URL_DECODE,2,pos + 1);
	new := CHR(DWORD_TO_BYTE(HEX_TO_DWORD(seq)));
	URL_DECODE := REPLACE(URL_DECODE, new, 3, pos);
	pos := FIND(URL_DECODE,'%');
END_WHILE;


(* revision history
hm		27. apr. 2008	rev 1.0
	original version

*)
END_FUNCTION

(* POU URL_ENCODE, ST *)
FUNCTION URL_ENCODE : STRING(255)
VAR_INPUT
	IN : STRING(255);
END_VAR
VAR
	pt_in : POINTER TO ARRAY[1..255] OF BYTE;
	pt_out : POINTER TO ARRAY[1..256] OF BYTE;
	pos_in : INT;
	pos_out : INT;
	stop : INT;
	tb : BYTE;
END_VAR


(*
version 1.0		27. apr. 2008
programmer 		hugo
tested by		hugo

URL_ENCODE checks a string if it contains only non reserved characters for an url.
the non reserved characters are : [A..Z], [a..z], [0..9], -_.~
if reserved characters are found then these characters are converted to %HH while HH is the Hexadezimal representation of the character in Alphabetic Letters.
for example the reserved character # will be converted to '%23'.

*)
pt_in  := ADR(in);
pt_out := ADR(URL_ENCODE);

(* scan the input string and convert unallowed characters *)
pos_in := 1;
stop := LEN(in);
FOR pos_out := 1 TO 255 DO
	IF pos_in > stop THEN
		EXIT;
	ELSIF IS_URLCHR(pt_in^[pos_in]) THEN
		pt_out^[pos_out] := pt_in^[pos_in];
		(* increment in by 1 *)
		pos_in := pos_in + 1;
	ELSE
		(* cannot fit 3 digits, exit *)
		IF pos_out > 253 THEN EXIT; END_IF;
		(* invalid character that needs to be converted *)
		pt_out^[pos_out] := 37;    (* start with % sign *)
		pos_out := pos_out + 1;
		(* need to add the two hex digits *)
		tb := SHR(pt_in^[pos_in],4);
		IF tb > 9 THEN
			pt_out^[pos_out] := tb + 55;
		ELSE
			pt_out^[pos_out] := tb + 48;
		END_IF;
		pos_out := pos_out + 1;
		tb := pt_in^[pos_in] AND 16#0F;
		IF tb > 9 THEN
			pt_out^[pos_out] := tb + 55;
		ELSE
			pt_out^[pos_out] := tb + 48;
		END_IF;
		(* increment in and out because out has to move 3 digits *)
		pos_in := pos_in + 1;
	END_IF;
END_FOR;

(* terminate the output string *)
pt_out^[pos_out] := 0;

(* revision history
hm		27. apr. 2008	rev 1.0
	original version

*)
END_FUNCTION

(* POU URL_TO_STRING, ST *)
FUNCTION URL_TO_STRING : STRING(255)
VAR_INPUT
	IN : URL;
END_VAR
VAR
END_VAR

(*
version 1.0	18. apr. 2008
programmer 	hugo
tested by		oscat

URL_TO_STRING generates a string from URL information suppied in IN..

*)
(*

http://hans:geheim@www.example.org:80/demo/example.cgi?land=de&stadt=aa#abschnitt1
|         |         |                  |                                |   |                                    |                                    |
|         |         |                 Host                         |   Pfad                            Query                           Anker
|         |         Passwort                                  Port
|        Benutzer
Protokoll

*)

(* attach protocol *)
IF IN.PROTOCOL <> '' THEN 	URL_TO_STRING := CONCAT(IN.PROTOCOL,'://'); END_IF;

(* attach user and password *)
IF IN.USER <> '' THEN
	URL_TO_STRING := CONCAT(URL_TO_STRING, IN.USER);
	IF IN.PASSWORD <> '' THEN
		URL_TO_STRING := CONCAT(URL_TO_STRING, ':');
		URL_TO_STRING := CONCAT(URL_TO_STRING, IN.PASSWORD);
	END_IF;
	URL_TO_STRING := CONCAT(URL_TO_STRING, '@');
END_IF;

(* attach domain *)
URL_TO_STRING := CONCAT(URL_TO_STRING, IN.DOMAIN);

(* attach Port *)
IF IN.PORT > 0 THEN
	URL_TO_STRING := CONCAT(URL_TO_STRING, ':');
	URL_TO_STRING := CONCAT(URL_TO_STRING, WORD_TO_STRING(IN.PORT));
END_IF;

(* attach path *)
URL_TO_STRING := CONCAT(URL_TO_STRING, IN.PATH);

(* attach query *)
IF IN.QUERY <> '' THEN
	URL_TO_STRING := CONCAT(URL_TO_STRING, '?');
	URL_TO_STRING := CONCAT(URL_TO_STRING, IN.QUERY);
END_IF;

(* attach anchor *)
IF IN.ANCHOR <> '' THEN
	URL_TO_STRING := CONCAT(URL_TO_STRING, '#');
	URL_TO_STRING := CONCAT(URL_TO_STRING, IN.ANCHOR);
END_IF;

(* revision history
hm		18. apr 2008	rev 1.0
	original version

*)
END_FUNCTION

(* POU V3_ABS, ST *)
FUNCTION V3_ABS : REAL
VAR_INPUT
	A : Vector_3;
END_VAR
VAR
END_VAR

(*
version 1.0	11 dec 2007
programmer 	hugo
tested by		tobias

this function calculates the length of a vectors in a 3 dimensional space

*)
V3_ABS := SQRT(A.X * A.X + A.Y * A.Y + A.Z * A.Z);


(* revision history
hm		11 dec 2007	rev 1.0
	original version

*)
END_FUNCTION

(* POU V3_ADD, ST *)
FUNCTION V3_ADD : vector_3
VAR_INPUT
	A : Vector_3;
	B : Vector_3;
END_VAR
VAR
END_VAR

(*
version 1.0	11 dec 2007
programmer 	hugo
tested by		tobias

this function adds two vectors in a 3 dimensional space

*)
V3_ADD.X := A.X + B.X;
V3_ADD.Y := A.Y + B.Y;
V3_ADD.Z := A.Z + B.Z;



(* revision history
hm		11 dec 2007	rev 1.0
	original version

*)
END_FUNCTION

(* POU V3_ANG, ST *)
FUNCTION V3_ANG : REAL
VAR_INPUT
	A : Vector_3;
	B : Vector_3;
END_VAR
VAR
	d : REAL;
END_VAR

(*
version 1.0	11 dec 2007
programmer 	hugo
tested by		tobias

this function calculates the angle between two vectors in a 3 dimensional space

*)
d := V3_ABS(A) * V3_ABS(B);
IF d > 0 THEN
	V3_ANG := ACOS(LIMIT(-1,V3_DPRO(A,B) / d,1));
END_IF;

(* revision history
hm		11 dec 2007	rev 1.0
	original version

*)
END_FUNCTION

(* POU V3_DPRO, ST *)
FUNCTION V3_DPRO : REAL
VAR_INPUT
	A : Vector_3;
	B : Vector_3;
END_VAR
VAR
END_VAR

(*
version 1.0	11 dec 2007
programmer 	hugo
tested by		tobias

this function calculates the dot product of two vectors in 3 dimensional space

*)
V3_DPRO := A.X * B.X + A.Y * B.Y + A.Z * B.Z;


(* revision history
hm		11 dec 2007	rev 1.0
	original version

*)
END_FUNCTION

(* POU V3_NORM, ST *)
FUNCTION V3_NORM : vector_3
VAR_INPUT
	A : Vector_3;
END_VAR
VAR
	la: REAL;
END_VAR

(*
version 1.0	11 dec 2007
programmer 	hugo
tested by		tobias

this function generates a vectors with absolute length 1 from a vector A in a 3 dimensional space

*)
la := V3_ABS(A);
IF la > 0 THEN
	V3_NORM := V3_SMUL(A,1/la);
END_IF;

(* revision history
hm		11 dec 2007	rev 1.0
	original version

*)
END_FUNCTION

(* POU V3_SMUL, ST *)
FUNCTION V3_SMUL : vector_3
VAR_INPUT
	A : Vector_3;
	M : REAL;
END_VAR
VAR
END_VAR

(*
version 1.0	11 dec 2007
programmer 	hugo
tested by		tobias

this function multiplies a vectors in a 3 dimensional space with a skalar M

*)
V3_SMUL.X := A.X * M;
V3_SMUL.Y := A.Y * M;
V3_SMUL.Z := A.Z * M;



(* revision history
hm		11 dec 2007	rev 1.0
	original version

*)
END_FUNCTION

(* POU V3_NUL, ST *)
FUNCTION V3_NUL : BOOL
VAR_INPUT
	A : Vector_3;
END_VAR
VAR
END_VAR

(*
version 1.0	12 dec 2007
programmer 	hugo
tested by		tobias

this function checks if a vectors in a null Vector

*)
V3_NUL := A.X = 0 AND A.Y = 0 AND A.Z = 0;



(* revision history
hm		12 dec 2007	rev 1.0
	original version

*)
END_FUNCTION

(* POU V3_PAR, ST *)
FUNCTION V3_PAR : BOOL
VAR_INPUT
	A : Vector_3;
	B : Vector_3;
END_VAR
VAR
END_VAR

(*
version 1.0	11 dec 2007
programmer 	hugo
tested by		tobias

this function checks if two vectors in a 3 dimensional space are parallel.
which means the two vectors have the same direction

*)
V3_PAR := V3_ABS(V3_XPRO(A,B)) = 0;



(* revision history
hm		11 dec 2007	rev 1.0
	original version

*)
END_FUNCTION

(* POU V3_XPRO, ST *)
FUNCTION V3_XPRO : vector_3
VAR_INPUT
	A : Vector_3;
	B : Vector_3;
END_VAR
VAR
END_VAR

(*
version 1.0	11 dec 2007
programmer 	hugo
tested by		tobias

this function adds two vectors in a 3 dimensional space

*)
V3_XPRO.X := A.Y * B.Z - A.Z * B.Y;
V3_XPRO.Y := A.Z * B.X - A.X * B.Z;
V3_XPRO.Z := A.X * B.Y - A.Y * B.X;



(* revision history
hm		11 dec 2007	rev 1.0
	original version

*)
END_FUNCTION

(* POU V3_REV, ST *)
FUNCTION V3_REV : vector_3
VAR_INPUT
	A : Vector_3;
END_VAR
VAR
END_VAR

(*
version 1.0	11 dec 2007
programmer 	hugo
tested by		tobias

this function reverses a vector in a 3 dimensional space

*)
V3_REV.X := -A.X;
V3_REV.Y := -A.Y;
V3_REV.Z := -A.Z;



(* revision history
hm		11 dec 2007	rev 1.0
	original version

*)
END_FUNCTION

(* POU V3_SUB, ST *)
FUNCTION V3_SUB : vector_3
VAR_INPUT
	A : Vector_3;
	B : Vector_3;
END_VAR
VAR
END_VAR

(*
version 1.0	11 dec 2007
programmer 	hugo
tested by		tobias

this function subtracts two vectors in a 3 dimensional space
V3_SUB = A - B

*)
V3_SUB.X := A.X - B.X;
V3_SUB.Y := A.Y - B.Y;
V3_SUB.Z := A.Z - B.Z;



(* revision history
hm		11 dec 2007	rev 1.0
	original version

*)
END_FUNCTION

(* POU V3_XANG, ST *)
FUNCTION V3_XANG : REAL
VAR_INPUT
	A : Vector_3;
END_VAR
VAR
	la: REAL;
END_VAR

(*
version 1.0	11 dec 2007
programmer 	hugo
tested by		tobias

this function calculates the angle between the X-axis and a vectors in a 3 dimensional space

*)
la := V3_ABS(a);
IF la > 0 THEN
	V3_XANG := ACOS(A.X / la);
END_IF;

(* revision history
hm		11 dec 2007	rev 1.0
	original version

*)
END_FUNCTION

(* POU V3_YANG, ST *)
FUNCTION V3_YANG : REAL
VAR_INPUT
	A : Vector_3;
END_VAR
VAR
	la: REAL;
END_VAR

(*
version 1.0	11 dec 2007
programmer 	hugo
tested by		tobias

this function calculates the angle between the Y-axis and a vectors in a 3 dimensional space

*)
la := V3_ABS(a);
IF la > 0 THEN
	V3_YANG := ACOS(A.Y / la);
END_IF;

(* revision history
hm		11 dec 2007	rev 1.0
	original version

*)
END_FUNCTION

(* POU V3_ZANG, ST *)
FUNCTION V3_ZANG : REAL
VAR_INPUT
	A : Vector_3;
END_VAR
VAR
	la: REAL;
END_VAR

(*
version 1.0	11 dec 2007
programmer 	hugo
tested by		tobias

this function calculates the angle between the Z-axis and a vectors in a 3 dimensional space

*)
la := V3_ABS(a);
IF la > 0 THEN
	V3_ZANG := ACOS(A.Z / la);
END_IF;

(* revision history
hm		11 dec 2007	rev 1.0
	original version

*)
END_FUNCTION

(* POU WATER_CP, ST *)
FUNCTION WATER_CP : REAL
VAR_INPUT
	T : REAL;
END_VAR
VAR
	Pts : INT := 10;
	data : ARRAY[1..20, 0..1] OF REAL := 0,4.228, 5,4.20, 10,4.188, 15,4.184, 50,4.181, 60,4.183, 70,4.187, 80,4.194, 90,4.204, 100,4.22;
END_VAR

(*
version 1.1	27 dec 2007 
programmer 	hugo
tested by	tobias

water_cp calculates the specific heat capacity of liquid water from 0..100 °C 

*)
water_CP := LINEAR_INT(T, Data, Pts);


(* revision history

hm	29.10.2007		rev 1.0
	original version

hm	27. dec 2007	rev 1.1
	increased accuracy

*)

(*
    °C - die Celsius-Temperatur in Grad Celsius
    v – das spezifische Volumen in Kubikdezimeter je Kilogramm dm³/kg
    h – die spezifische Enthalpie in Kilojoule je Kilogramm 	kJ/kg
    u – die spezifische Innere Energie in Kilojoule je Kilogramm 	kJ/kg
    s – die spezifische Entropie in Kilojoule je Kilogramm mal Kelvin 	kJ/(kg·K)
    cp - die spezifische Wärmekapazität bei konstantem Druck in Kilojoule je Kilogramm mal Kelvin 	kJ/(kg·K)
    Y – Volumenausdehnungskoeffizient in 10-3 durch Kelvin  10-3/K
    L – Wärmeleitfähigkeit in Milliwatt je Meter mal Kelvin  mW / (m·K) 
    n – Viskosität in Mikropascal mal Sekunde uPa·s 	
    s ? – Oberflächenspannung in Millinewton je Meter  mN/m


°C 		v 				h 			u 		s 			cp 		Y 		L		n		s	
-20		1,006580	
0 		1,000160 		0,06 		-0,04 	-0,0001 	4,228 	-0,080 	561,0 	1792 	75,65
4		1,000028
5 		1,0000 		21,1 		21,0 	0,076 		4,200 	0,011 	570,6 	1518 	74,95
10 		1,0003 		42,1 		42,0 	0,151 		4,188 	0,087 	580,0 	1306 	74,22
15 		1,0009 		63,0 		62,9 	0,224 		4,184 	0,152 	589,4 	1137 	73,49
20 		1,001797 		83,9 		83,8 	0,296 		4,183 	0,209 	598,4 	1001 	72,74
25 		1,0029 		104,8 		104,7 	0,367 		4,183 	0,259 	607,2 	890,4 	71,98
30 		1,0044 		125,8 		125,7 	0,437 		4,183 	0,305 	615,5 	797,7 	71,20
35 		1,0060 		146,7 		146,6 	0,505 		4,183 	0,347 	623,3 	719,6 	70,41
40 		1,007842 		167,58 	167,5 	0,572 		4,182 	0,386 	630,6 	653,3 	69,60
45 		1,0099 		188,5 		188,4 	0,638 		4,182 	0,423 	637,3 	596,3 	68,78
50 		1,0121 		209,4 		209,3 	0,704 		4,181 	0,457 	643,6 	547,1 	67,95
60 		1,017089 		251,2 		251,1 	0,831 		4,183 	0,522 	654,4 	466,6 	66,24
70 		1,0227 		293,1 		293,0 	0,955 		4,187 	0,583 	663,1 	404,1 	64,49
80 		1,029027 		335,0 		334,9 	1,075 		4,194 	0,640 	670,0 	354,5 	62,68
90 		1,0359 		377,0 		376,9 	1,193 		4,204 	0,696 	675,3 	314,6 	60,82
99,63 	1,0431 		417,5 		417,4 	1,303 		4,217 	0,748 	679,0 	283,0 	58,99
100	1,043453		419,1

Stoffdaten von Wasser Quelle Wickipedia

Wasser hat unter Normaldruck seine größte Dichte von 1000 Kilogramm pro Kubikmeter bei 3,98 °C und zeigt damit eine Dichteanomalie. 
Diese besteht darin, dass sich Wasser unterhalb von 3,98 °C bei weiterer Temperaturverringerung, auch beim Wechsel zum festen 
Aggregatzustand, wieder ausdehnt, was man nur von wenigen Stoffen kennt. Die derzeit genauesten publizierten Werte für die maximale 
Dichte liegen bei (999,974950 ± 0,00084) kg/m³ und bei (3,983 ± 0,00067) °C für die Temperatur, bei der dieser Wert erreicht wird. 
Die Werte stellen einen Mittelwert der von verschiedenen physikalischen Instituten veröffentlichten Zahlen dar (Stand 2001).

Die Berechnung der Dichte von luftfreiem Wasser DLF in Abhängigkeit von der Temperatur T ([T] = °C) kann mit Hilfe der folgenden 
Virialgleichung erfolgen:
: \frac{D_{\rm LF}}{\rm g/l} = \frac{a_0 + a_1 T + a_2 T^2 + a_3 T^3 + a_4 T^4 + a_5 T^5}{1 + b T}.
mit den Koeffizienten: a0 = 999,83952; a1 = 16,952577 (°C)-1; a2 = -7,9905127·10-3 (°C)-2; a3 = -4,6241757·10-5 (°C)-3; 
a4 = 1,0584601·10-7 (°C)-4; a5 = -2,8103006·10-10 (°C)-5 und b = 0,0168872. 
Für die Berechnung der Dichte von luftgesättigtem Wasser korrigiert man den Wert nach 
DLG/(g/l) = DLF/(g/l) - 0,004612 + 0,000106 (°C)-1·T. (Quelle: PTB-Mitteilungen 100/3-90)

*)
END_FUNCTION

(* POU WCT, ST *)
FUNCTION WCT : REAL
VAR_INPUT
	T : REAL;
	V : REAL;
END_VAR
VAR
END_VAR

(*
version 1.1	7 dec 2007
programmer 	hugo
tested by		tobias

this function calculates the wind chill temperature

*)
IF V < 5 OR T > 10 THEN
	WCT := T;
ELSE
	WCT := 13.12 + 0.6215 * T +(0.3965 * T - 11.37) * EXP(LN(v) * 0.16);
END_IF;


(* revision history
hm		7 feb 2007
	original version

hm		7 dec 2007
	changed code for better performance

*)
END_FUNCTION

(* POU WINDOW, ST *)
FUNCTION WINDOW : BOOL
VAR_INPUT
	low : REAL;
	in : REAL;
	high : REAL;
END_VAR
VAR
END_VAR

(*
	version 1.1	22 jan 2007
	programmer 	hugo
	tested BY	tobias

this checks a signal if the signal is between the upper and lower limit
*)
WINDOW := in < high AND in > low;


(* revision history
hm	22.1.2007	rev 1.1
	changed the order of inputs to low, in, high

*)
END_FUNCTION

(* POU WINDOW2, ST *)
FUNCTION WINDOW2 : BOOL
VAR_INPUT
	low : REAL;
	in : REAL;
	high : REAL;
END_VAR
VAR
END_VAR

(*
	version 1.0	31 oct 2007
	programmer 	hugo
	tested BY	tobias

this checks a signal if the signal is between the upper and lower limit including the two limits
*)
WINDOW2 := in <= high AND in >= low;


(* revision history
hm	31.10.2007	rev 1.0
	original version

*)
END_FUNCTION

(* POU WORD_OF_BYTE, ST *)
FUNCTION WORD_OF_BYTE : WORD
VAR_INPUT
	B1 : BYTE;
	B0 : BYTE;
END_VAR
VAR
END_VAR

(*
version 1.3	23. apr. 2008
programmer 	hugo
tested by		tobias

this function creates a word from 2 individual bytes

*)
WORD_OF_BYTE := SHL(B1,8) OR B0;

(* revision history
hm	24. jan 2007	rev 1.0
	original version

hm	2. jan 2008	rev 1.1
	improved performance

hm	19. feb 2008	rev 1.2
	replaced and with or for better compatibility

hm	23. apr. 2008	rev 1.3
	reverse order of inputs to be more logical
*)
END_FUNCTION

(* POU WORD_OF_DWORD, ST *)
FUNCTION WORD_OF_DWORD : WORD
VAR_INPUT
	in : DWORD;
	N : BYTE;
END_VAR
VAR
END_VAR

(*
version 1.1	2 jan 2008
programmer 	hugo
tested by		tobias

this function extracts a single word from the nth position from right (right is lowest byte)
the lower word (starting with Bit0 from in) is selected with N=0.
*)
Word_of_Dword := DWORD_TO_WORD(SHR(in,n*16));

(* revision history
hm	17. jan 2007	rev 1.0
	original version

hm	2. jan 2008		rev 1.1
	improved performance

*)
END_FUNCTION

(* POU WORD_TO_RANGE, ST *)
FUNCTION WORD_TO_RANGE : REAL
VAR_INPUT
	X : WORD;
	low : REAL;
	high : REAL;
END_VAR
VAR
END_VAR

(*
version 1.0	9. jan 2008
programmer 	hugo
tested by		tobias

Word_to_Range converts a Byte into a real between low and high.

*)
Word_to_Range := (high - low) * X / 65535.0 + low;


(* revision history
hm	9. jan 2008		rev 1.0
	original version

*)
END_FUNCTION

(* POU WORK_WEEK, ST *)
FUNCTION WORK_WEEK : INT
VAR_INPUT
	idate : DATE;
END_VAR
VAR
	d1 : DATE;
	w1 : INT;
	ds: DWORD;
	yr: INT;
	w31: INT;
	w01: INT;
	wm: INT;
END_VAR

(*
version 1.3	16 mar 2008
programmer 	hugo
tested by		tobias

calculates the work week for a given date according to iso8601

*)
(* berechne den 1.1 des jahres von idate. *)
yr := year(idate);
d1 := year_begin(yr);
(* wochentag von d1 *)
w1 := weekday(d1);
(* offset des montags der eletzten KW des vorjahres *)
(* wenn der erste tag des jahres größer als donnerstag ist dann beginnt die letzte kw am montag davor *)
(* wenn der erste tag des jahres ein donnerstag oder kleiner ist beginnt die erste kw 2 montage davor *)
IF w1 < 5 THEN
	ds := DATE_TO_DWORD(d1) - INT_TO_DWORD(w1+6) * 86400;
ELSE
	ds := DATE_TO_DWORD(d1) - INT_TO_DWORD(w1-1) * 86400;
END_IF;

(* kalenderwoche des eingangsdatums *)
work_week := DWORD_TO_INT((DATE_TO_DWORD(idate) - ds) / 604800);

(* korrektur wenn work_week = 0 *)
IF work_week = 0 THEN
	(* work_week needs to be 53 when 1.jan of the year before is thursday or dec 31. is thursday. *)
	(* first and last weekday of a year is equal and one more day for a leap_year. *)
	IF w1 > 1 THEN w31 := w1 - 1; ELSE W31 := 7; END_IF;
	IF leap_year(yr - 1) THEN IF w31 > 1 THEN w01 := W31 - 1; ELSE w1 := 7; END_IF; END_IF;
	(* if first or last day of a year is a thursday, the year has 53 weeks *)
	IF w31 = 4 OR w01 = 4 THEN work_week := 53; ELSE work_week := 52; END_IF;
ELSE
	(* end of year calculation *)
	(* calculated the first and last weekday *)
	IF leap_year(yr) THEN
		IF w1 < 7 THEN w31 := w1 + 1; ELSE w31 := 1; END_IF;
	ELSE
		w31 := w1;
	END_IF;
	(* if first or last day is thursday then the year has 53 weeks otherwise only 52 *)
	IF w31 = 4 OR w1 = 4 THEN wm := 53; ELSE wm := 52; END_IF;
	IF work_week > wm THEN work_week := 1; END_IF;
END_IF;



(* old code before rev 1.2
w1 := weekday(set_Date(year(idate), 1,1));
IF w1 < 5 THEN
	work_week := (day_of_year(idate) + w1 + 5)/7;
ELSE
	work_week := (day_of_year(idate) + w1 - 2)/7;
END_IF
*)


(* revision history

hm 17.1.2007		rev 1.1
	deleted unused variable yday

hm	19. dec 2007	rev 1.2
	changed code for better performance
	changed code to comply with ISO8601

hm	16. mar 2008	rev 1.3
	added type conversions to avoid warnings under codesys 3.0
*)
END_FUNCTION
